{attribute addProperty BoxType "KL6211"}
{attribute addProperty Id "Channel_1Channel_A455ADD900"}
{attribute addProperty CRC "2450587506"}
{attribute addProperty SizeInBites "0"}
{attribute addProperty SizeInBytes "0"}
TYPE KL6211_9210FF72 :
STRUCT
	{attribute addProperty Name "Channel_1"}
	Channel_1 : Channel_A455ADD9;
END_STRUCT
END_TYPE

(* stored: Version 1.2.0.0, ProductVersion 3.1.4024.9
   DUT KL6211_9210FF72: Id {46bb73aa-7be5-4b1a-b06c-74da5b31dbb2} *)
